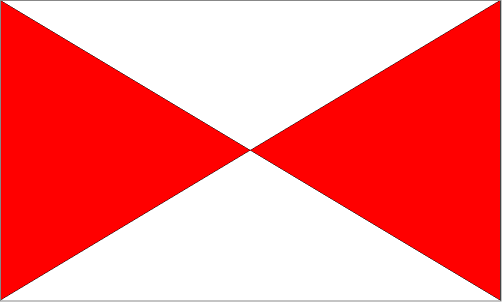
VISUALIZATION visuFCVSim  // 502x302
    Polygon (0,0) (0,300) (250,150), invisible if: NOT progFCVCntrl.FCV_04_0100.FB_Close
    Polygon (500,0) (500,300) (250,150), invisible if: NOT progFCVCntrl.FCV_04_0100.FB_Close
    Polygon (0,0) (0,300) (250,150), invisible if: NOT progFCVCntrl.FCV_04_0100.FB_Travelling
    Polygon (500,0) (500,300) (250,150), invisible if: NOT progFCVCntrl.FCV_04_0100.FB_Travelling
    Polygon (0,0) (0,300) (250,150), invisible if: NOT progFCVCntrl.FCV_04_0100.FB_Open
    Polygon (500,0) (500,300) (250,150), invisible if: NOT progFCVCntrl.FCV_04_0100.FB_Open
    Polygon (0,0) (0,300) (250,150), invisible if: NOT progFCVCntrl.FCV_04_0100.Alarm
    Polygon (500,0) (500,300) (250,150), invisible if: NOT progFCVCntrl.FCV_04_0100.Alarm
END_VISUALIZATION

(* stored: Version 1.1.0.1, ProductVersion 3.1.4022.17
   Visu visuFCVSim: Id {5fe1c757-3858-479a-b1c8-78ca66ebe74a} *)
